{attribute 'qualified_only'}
VAR_GLOBAL
	// Simulation IHM
	StartSystem: BOOL;
	StopSystem: BOOL;

END_VAR

(* stored: Version 1.1.0.1, ProductVersion 3.1.4024.11
   GVL GVL_IHM: Id {ab0fb600-c17b-467c-8d8f-d7596e54b9a2} *)
